PROGRAM POU
VAR
END_VAR

// NETWORK 1

END_PROGRAM

(* stored: Version 1.1.0.1, ProductVersion 3.1.4024.13
   POU POU: Id {e9f9ce50-05c7-47e4-8732-1d2fd1c06e2e}, SpecialFunc None *)
